// TIA Portal V20 export
TYPE "typeFDoorFunction"
// Safety status of door
// stored: Access Published, IsFailsafeCompliant true, Namespace Safety
   STRUCT
      fDoor1 : "Safety.typeFDoorFunctionData";
      fDoor2 : "Safety.typeFDoorFunctionData";
      fDoor3 : "Safety.typeFDoorFunctionData";
      fDoor4 : "Safety.typeFDoorFunctionData";
      fDoor5 : "Safety.typeFDoorFunctionData";
      fDoor6 : "Safety.typeFDoorFunctionData";
      fDoor7 : "Safety.typeFDoorFunctionData";
      fDoor8 : "Safety.typeFDoorFunctionData";
      fDoor9 : "Safety.typeFDoorFunctionData";
      fDoor10 : "Safety.typeFDoorFunctionData";
   END_STRUCT;
END_TYPE
